TYPE T_Ctrl_SIf_MOD_DtChnToPLC :
STRUCT
	dinTest : DINT;
	intDataState : INT;
END_STRUCT
END_TYPE

(* stored: Version 1.1.0.1, ProductVersion 3.1.0.19
   DUT T_Ctrl_SIf_MOD_DtChnToPLC: Id {6431b662-259f-4c30-bb7c-d3235bf970f0} *)
